// TIA Portal project "Calculate" (V17)

(* hardware
DEVICE "S7-1200 station_1"  S7-1200 Station
   slot 0: "Rack_0"  S7-1200 Rack  Rack  V1.0
   slot 1: "PLC_1"  CPU 1212C DC/DC/DC  6ES7 212-1AE40-0XB0  V4.5
*)

// ===== PLC "PLC_1"  CPU 1212C DC/DC/DC =====

DATA_BLOCK "Calculate_DB"   // DB1
{ S7_Optimized_Access := 'TRUE' }
VERSION : 0.1
   VAR
      Power : Struct
         Int_a : Int;
         Int_b : Int;
         Int_c : Int;
      END_STRUCT;
      ADD : Struct
         Int_a : Int;
         Int_b : Int;
         Int_c : Int;
      END_STRUCT;
      SUB : Struct
         Int_a : Int;
         Int_b : Int;
         Int_c : Int;
      END_STRUCT;
      MUL : Struct
         Int_a : Int;
         Int_b : Int;
         Int_c : Int;
      END_STRUCT;
      DIV : Struct
         Int_a : Int;
         Int_b : Int;
         Int_c : Int;
      END_STRUCT;
      Calculate : Struct
         Int_a_Input : Int;
         Int_b_Input : Int;
         Int_c_Input : Int;
         Int_d_Output : Real;
      END_STRUCT;
   END_VAR
BEGIN
END_DATA_BLOCK

FUNCTION "Test One" : Void   // FC1, SCL
{ S7_Optimized_Access := 'TRUE' }
VERSION : 0.1
BEGIN
   //幂运算 Power
   "Calculate_DB".Power.Int_c := "Calculate_DB".Power.Int_b ** "Calculate_DB".Power.Int_a;

   //加法运算 ADD
   "Calculate_DB".ADD.Int_c := "Calculate_DB".ADD.Int_b + "Calculate_DB".ADD.Int_a;

   //减法运算 SUB
   "Calculate_DB".SUB.Int_c := "Calculate_DB".SUB.Int_b - "Calculate_DB".SUB.Int_a;

   //乘法运算 MUL
   "Calculate_DB".MUL.Int_c := "Calculate_DB".MUL.Int_b * "Calculate_DB".MUL.Int_a;

   //除法运算 DIV
   "Calculate_DB"."DIV".Int_c := "Calculate_DB"."DIV".Int_b / "Calculate_DB"."DIV".Int_a;

   //计算 a+(b*c) 在进行幂运算 **2 再 /4 Calculate
   "Calculate_DB".Calculate.Int_d_Output := (("Calculate_DB".Calculate.Int_c_Input * "Calculate_DB".Calculate.Int_b_Input) + "Calculate_DB".Calculate.Int_a_Input) ** 2 / 4;
END_FUNCTION

ORGANIZATION_BLOCK "Main"   // OB1, LAD, ProgramCycle
TITLE = "Main Program Sweep (Cycle)"
{ S7_Optimized_Access := 'TRUE' }
VERSION : 0.1
   VAR_INPUT
      Initial_Call : Bool;   // Initial call of this OB
      Remanence : Bool;   // =True, if remanent data are available
   END_VAR
BEGIN

REGION Network 1
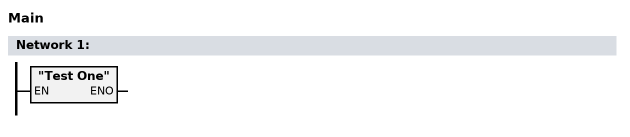
   RUNG wire#powerrail
      "Test One"()
   END_RUNG
   // the same network as SCL:
   "Test One"();
END_REGION
END_ORGANIZATION_BLOCK